PROGRAM automat_PRG
VAR_INPUT
SFCInit: BOOL; 
END_VAR
VAR
	counter: INT; //counting cyklus
END_VAR

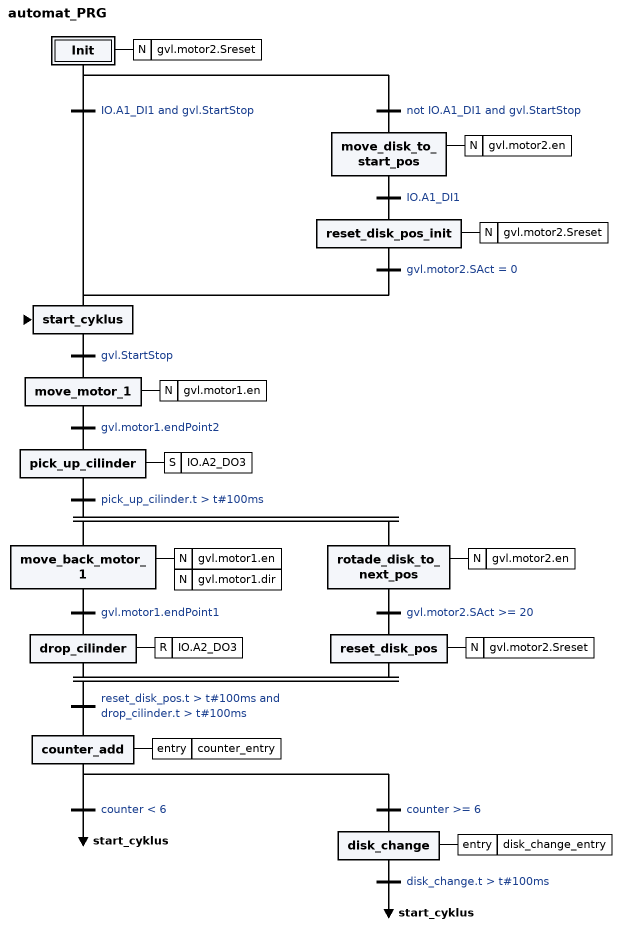
INITIAL_STEP Init:
    gvl.motor2.Sreset(N);
END_STEP
TRANSITION FROM Init TO start_cyklus
    := IO.A1_DI1 and gvl.StartStop;
END_TRANSITION
TRANSITION FROM Init TO move_disk_to_start_pos
    := not IO.A1_DI1 and gvl.StartStop;
END_TRANSITION
STEP move_disk_to_start_pos:
    gvl.motor2.en(N);
END_STEP
TRANSITION FROM move_disk_to_start_pos TO reset_disk_pos_init
    := IO.A1_DI1;
END_TRANSITION
STEP reset_disk_pos_init:
    gvl.motor2.Sreset(N);
END_STEP
TRANSITION FROM reset_disk_pos_init TO start_cyklus
    := gvl.motor2.SAct = 0;
END_TRANSITION
STEP start_cyklus:
END_STEP
TRANSITION FROM start_cyklus TO move_motor_1
    := gvl.StartStop;
END_TRANSITION
STEP move_motor_1:
    gvl.motor1.en(N);
END_STEP
TRANSITION FROM move_motor_1 TO pick_up_cilinder
    := gvl.motor1.endPoint2;
END_TRANSITION
STEP pick_up_cilinder:
    IO.A2_DO3(S);
END_STEP
TRANSITION FROM pick_up_cilinder TO (move_back_motor_1, rotade_disk_to_next_pos)
    := pick_up_cilinder.t > t#100ms;
END_TRANSITION
STEP move_back_motor_1:
    gvl.motor1.en(N);
    gvl.motor1.dir(N);
END_STEP
TRANSITION FROM move_back_motor_1 TO drop_cilinder
    := gvl.motor1.endPoint1;
END_TRANSITION
STEP drop_cilinder:
    IO.A2_DO3(R);
END_STEP
STEP rotade_disk_to_next_pos:
    gvl.motor2.en(N);
END_STEP
TRANSITION FROM rotade_disk_to_next_pos TO reset_disk_pos
    := gvl.motor2.SAct >= 20;
END_TRANSITION
STEP reset_disk_pos:
    gvl.motor2.Sreset(N);
END_STEP
TRANSITION FROM (drop_cilinder, reset_disk_pos) TO counter_add
    := reset_disk_pos.t > t#100ms and drop_cilinder.t > t#100ms;
END_TRANSITION
STEP counter_add:
    counter_entry(P1);  // entry action
END_STEP
TRANSITION FROM counter_add TO start_cyklus
    := counter < 6;
END_TRANSITION
TRANSITION FROM counter_add TO disk_change
    := counter >= 6;
END_TRANSITION
STEP disk_change:
    disk_change_entry(P1);  // entry action
END_STEP
TRANSITION FROM disk_change TO start_cyklus
    := disk_change.t > t#100ms;
END_TRANSITION

ACTION counter_entry:
counter := counter + 1;
END_ACTION

ACTION disk_change_entry:
counter := 0;
END_ACTION

END_PROGRAM

(* stored: Version 1.1.0.1, ProductVersion 3.1.4024.12
   POU automat_PRG: Id {6c22cb57-c4c2-44cd-9077-a0782cc89254}, SpecialFunc None
   Action counter_entry: Id {9eea2d37-9bf4-406a-b474-2974c3a7790b}
   Action disk_change_entry: Id {606da4a9-a278-4a6f-92d8-8a43f7fa7c71} *)
